FUNCTION_BLOCK FB_BaseGroupElement_HMI EXTENDS FB_BaseControlElement_HMI IMPLEMENTS ITF_BaseGroupElement_HMI
VAR
	itfBaseGroupElementConnector		: ITF_BaseGroupElement_HMI_Connector;
	refstBaseGroupElementDataHMI		: REFERENCE TO ST_BaseGroupElement_HMI;
	(*	lista elementów składających się na ten element w elemencie docelowym dodać itf dla konkretnych elementów	*)
	arrControlElement					: ARRAY [1..GVL_BaseConstans.MAX_ITEM_PER_ELEMENT] OF ITF_BaseControlElement_HMI;
	uiNumberOfControlElement			: UINT;
END_VAR

METHOD PROTECTED AddControlElement : BOOL
VAR_INPUT
	itfControlElementHMI		: ITF_BaseControlElement_HMI;
END_VAR
IF (THIS^.uiNumberOfControlElement + 1 <= GVL_BaseConstans.MAX_ITEM_PER_ELEMENT) THEN
	THIS^.uiNumberOfControlElement		:= THIS^.uiNumberOfControlElement + 1;
	THIS^.arrControlElement [THIS^.uiNumberOfControlElement]	:= itfControlElementHMI;
	AddControlElement			:= TRUE;
ELSE
	;//zwrocenie zbyt dużo komponentow
END_IF
END_METHOD

END_FUNCTION_BLOCK

(* stored: Version 1.1.0.1
   POU FB_BaseGroupElement_HMI: Id {3f198324-9925-0fb3-39d4-b6620e2a327f}, SpecialFunc None
   Method AddControlElement: Id {76a032d3-46d3-05c1-2da2-40ea71aff009} *)
